{attribute 'qualified_only'}
VAR_GLOBAL
	result : STRING(30);
END_VAR

(* stored: Version 1.1.0.1, ProductVersion 3.1.4024.16
   GVL GVL: Id {1c0c5ac1-78ac-4977-a7d6-da996df388f7} *)
